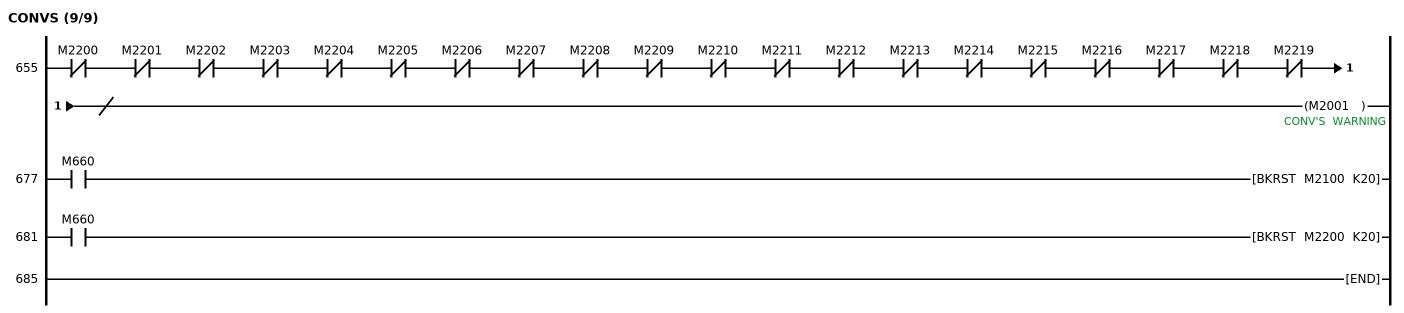
[picture p24: ladder of CONVS, rungs at steps 655 to 685]
655   LDI     M2200
      ANI     M2201
      ANI     M2202
      ANI     M2203
      ANI     M2204
      ANI     M2205
      ANI     M2206
      ANI     M2207
      ANI     M2208
      ANI     M2209
      ANI     M2210
      ANI     M2211
      ANI     M2212
      ANI     M2213
      ANI     M2214
      ANI     M2215
      ANI     M2216
      ANI     M2217
      ANI     M2218
      ANI     M2219
      INV
      OUT     M2001  ; CONV'S  WARNING
677   LD      M660
      BKRST   M2100 K20
681   LD      M660
      BKRST   M2200 K20
685   END
END_PROGRAM

PROGRAM CONV1
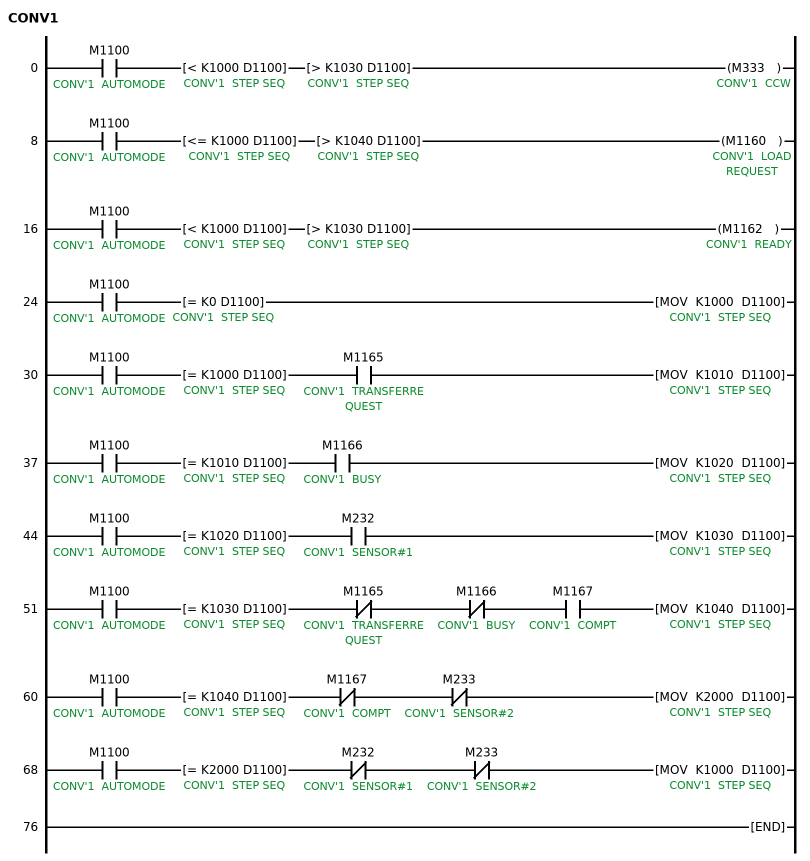
0     LD      M1100  ; CONV'1  AUTOMODE
      AND<    K1000 D1100  ; CONV'1  STEP SEQ
      AND>    K1030 D1100  ; CONV'1  STEP SEQ
      OUT     M333  ; CONV'1  CCW
8     LD      M1100  ; CONV'1  AUTOMODE
      AND<=   K1000 D1100  ; CONV'1  STEP SEQ
      AND>    K1040 D1100  ; CONV'1  STEP SEQ
      OUT     M1160  ; CONV'1  LOAD    REQUEST
16    LD      M1100  ; CONV'1  AUTOMODE
      AND<    K1000 D1100  ; CONV'1  STEP SEQ
      AND>    K1030 D1100  ; CONV'1  STEP SEQ
      OUT     M1162  ; CONV'1  READY
24    LD      M1100  ; CONV'1  AUTOMODE
      AND=    K0 D1100  ; CONV'1  STEP SEQ
      MOV     K1000 D1100
30    LD      M1100  ; CONV'1  AUTOMODE
      AND=    K1000 D1100  ; CONV'1  STEP SEQ
      AND     M1165  ; CONV'1  TRANSFERREQUEST
      MOV     K1010 D1100
37    LD      M1100  ; CONV'1  AUTOMODE
      AND=    K1010 D1100  ; CONV'1  STEP SEQ
      AND     M1166  ; CONV'1  BUSY
      MOV     K1020 D1100
44    LD      M1100  ; CONV'1  AUTOMODE
      AND=    K1020 D1100  ; CONV'1  STEP SEQ
      AND     M232  ; CONV'1  SENSOR#1
      MOV     K1030 D1100
51    LD      M1100  ; CONV'1  AUTOMODE
      AND=    K1030 D1100  ; CONV'1  STEP SEQ
      ANI     M1165  ; CONV'1  TRANSFERREQUEST
      ANI     M1166  ; CONV'1  BUSY
      AND     M1167  ; CONV'1  COMPT
      MOV     K1040 D1100
60    LD      M1100  ; CONV'1  AUTOMODE
      AND=    K1040 D1100  ; CONV'1  STEP SEQ
      ANI     M1167  ; CONV'1  COMPT
      ANI     M233  ; CONV'1  SENSOR#2
      MOV     K2000 D1100
68    LD      M1100  ; CONV'1  AUTOMODE
      AND=    K2000 D1100  ; CONV'1  STEP SEQ
      ANI     M232  ; CONV'1  SENSOR#1
      ANI     M233  ; CONV'1  SENSOR#2
      MOV     K1000 D1100
76    END
END_PROGRAM

PROGRAM CONV2
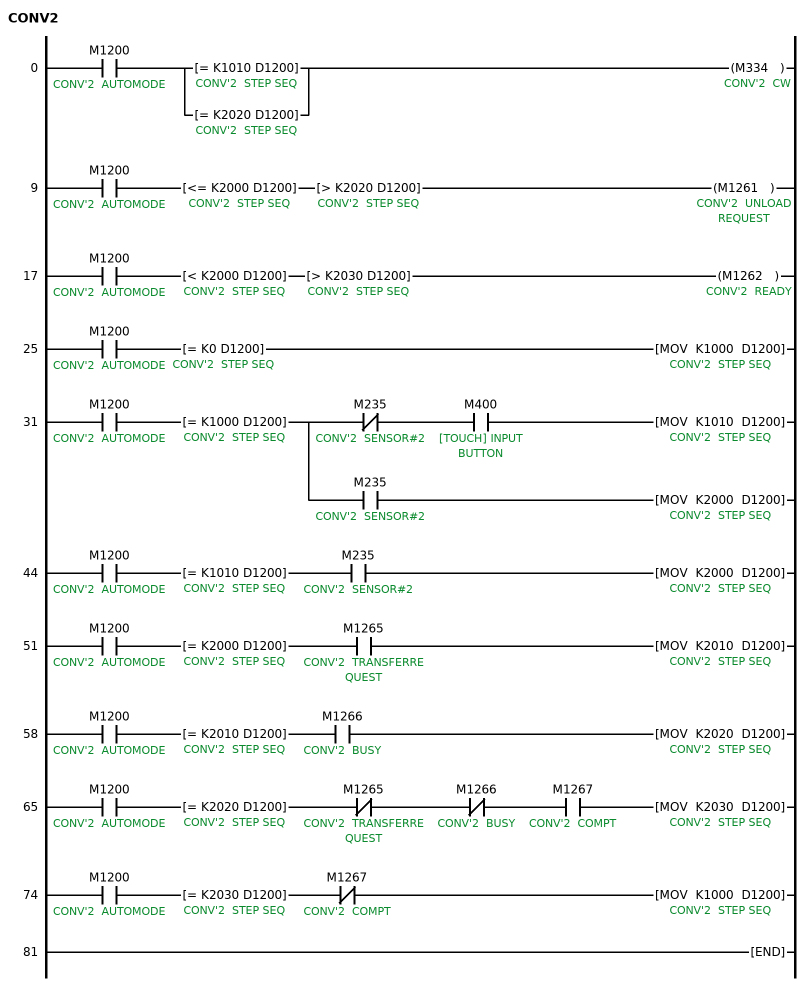
0     LD      M1200  ; CONV'2  AUTOMODE
      LD=     K1010 D1200  ; CONV'2  STEP SEQ
      OR=     K2020 D1200  ; CONV'2  STEP SEQ
      ANB
      OUT     M334  ; CONV'2  CW
9     LD      M1200  ; CONV'2  AUTOMODE
      AND<=   K2000 D1200  ; CONV'2  STEP SEQ
      AND>    K2020 D1200  ; CONV'2  STEP SEQ
      OUT     M1261  ; CONV'2  UNLOAD  REQUEST
17    LD      M1200  ; CONV'2  AUTOMODE
      AND<    K2000 D1200  ; CONV'2  STEP SEQ
      AND>    K2030 D1200  ; CONV'2  STEP SEQ
      OUT     M1262  ; CONV'2  READY
25    LD      M1200  ; CONV'2  AUTOMODE
      AND=    K0 D1200  ; CONV'2  STEP SEQ
      MOV     K1000 D1200
31    LD      M1200  ; CONV'2  AUTOMODE
      AND=    K1000 D1200  ; CONV'2  STEP SEQ
      MPS
      ANI     M235  ; CONV'2  SENSOR#2
      AND     M400  ; [TOUCH] INPUT   BUTTON
      MOV     K1010 D1200
      MPP
      AND     M235  ; CONV'2  SENSOR#2
      MOV     K2000 D1200
44    LD      M1200  ; CONV'2  AUTOMODE
      AND=    K1010 D1200  ; CONV'2  STEP SEQ
      AND     M235  ; CONV'2  SENSOR#2
      MOV     K2000 D1200
51    LD      M1200  ; CONV'2  AUTOMODE
      AND=    K2000 D1200  ; CONV'2  STEP SEQ
      AND     M1265  ; CONV'2  TRANSFERREQUEST
      MOV     K2010 D1200
58    LD      M1200  ; CONV'2  AUTOMODE
      AND=    K2010 D1200  ; CONV'2  STEP SEQ
      AND     M1266  ; CONV'2  BUSY
      MOV     K2020 D1200
65    LD      M1200  ; CONV'2  AUTOMODE
      AND=    K2020 D1200  ; CONV'2  STEP SEQ
      ANI     M1265  ; CONV'2  TRANSFERREQUEST
      ANI     M1266  ; CONV'2  BUSY
      AND     M1267  ; CONV'2  COMPT
      MOV     K2030 D1200
74    LD      M1200  ; CONV'2  AUTOMODE
      AND=    K2030 D1200  ; CONV'2  STEP SEQ
      ANI     M1267  ; CONV'2  COMPT
      MOV     K1000 D1200
81    END
END_PROGRAM

PROGRAM CONV3
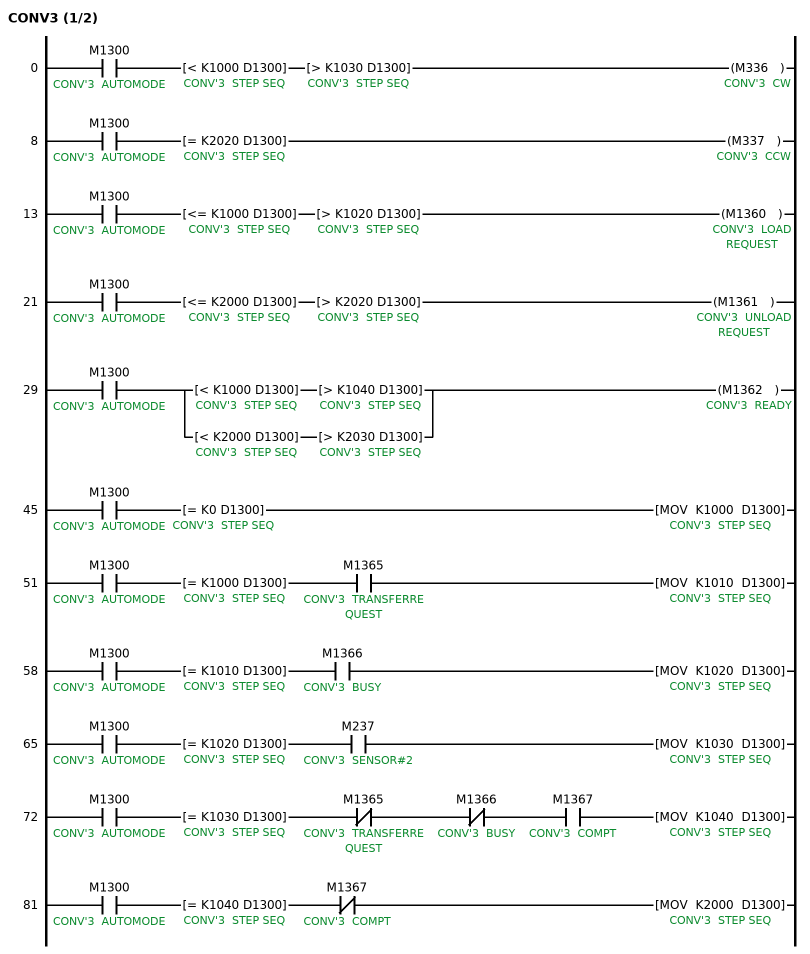
0     LD      M1300  ; CONV'3  AUTOMODE
      AND<    K1000 D1300  ; CONV'3  STEP SEQ
      AND>    K1030 D1300  ; CONV'3  STEP SEQ
      OUT     M336  ; CONV'3  CW
8     LD      M1300  ; CONV'3  AUTOMODE
      AND=    K2020 D1300  ; CONV'3  STEP SEQ
      OUT     M337  ; CONV'3  CCW
13    LD      M1300  ; CONV'3  AUTOMODE
      AND<=   K1000 D1300  ; CONV'3  STEP SEQ
      AND>    K1020 D1300  ; CONV'3  STEP SEQ
      OUT     M1360  ; CONV'3  LOAD    REQUEST
21    LD      M1300  ; CONV'3  AUTOMODE
      AND<=   K2000 D1300  ; CONV'3  STEP SEQ
      AND>    K2020 D1300  ; CONV'3  STEP SEQ
      OUT     M1361  ; CONV'3  UNLOAD  REQUEST
29    LD      M1300  ; CONV'3  AUTOMODE
      LD<     K1000 D1300  ; CONV'3  STEP SEQ
      AND>    K1040 D1300  ; CONV'3  STEP SEQ
      LD<     K2000 D1300  ; CONV'3  STEP SEQ
      AND>    K2030 D1300  ; CONV'3  STEP SEQ
      ORB
      ANB
      OUT     M1362  ; CONV'3  READY
45    LD      M1300  ; CONV'3  AUTOMODE
      AND=    K0 D1300  ; CONV'3  STEP SEQ
      MOV     K1000 D1300
51    LD      M1300  ; CONV'3  AUTOMODE
      AND=    K1000 D1300  ; CONV'3  STEP SEQ
      AND     M1365  ; CONV'3  TRANSFERREQUEST
      MOV     K1010 D1300
58    LD      M1300  ; CONV'3  AUTOMODE
      AND=    K1010 D1300  ; CONV'3  STEP SEQ
      AND     M1366  ; CONV'3  BUSY
      MOV     K1020 D1300
65    LD      M1300  ; CONV'3  AUTOMODE
      AND=    K1020 D1300  ; CONV'3  STEP SEQ
      AND     M237  ; CONV'3  SENSOR#2
      MOV     K1030 D1300
72    LD      M1300  ; CONV'3  AUTOMODE
      AND=    K1030 D1300  ; CONV'3  STEP SEQ
      ANI     M1365  ; CONV'3  TRANSFERREQUEST
      ANI     M1366  ; CONV'3  BUSY
      AND     M1367  ; CONV'3  COMPT
      MOV     K1040 D1300
81    LD      M1300  ; CONV'3  AUTOMODE
      AND=    K1040 D1300  ; CONV'3  STEP SEQ
      ANI     M1367  ; CONV'3  COMPT
      MOV     K2000 D1300
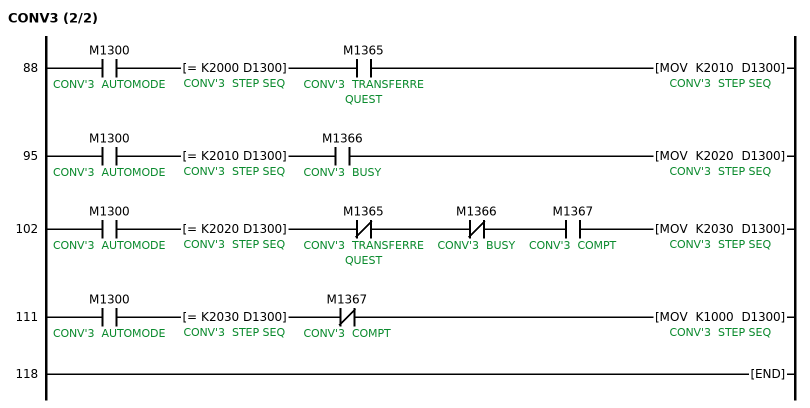
88    LD      M1300  ; CONV'3  AUTOMODE
      AND=    K2000 D1300  ; CONV'3  STEP SEQ
      AND     M1365  ; CONV'3  TRANSFERREQUEST
      MOV     K2010 D1300
95    LD      M1300  ; CONV'3  AUTOMODE
      AND=    K2010 D1300  ; CONV'3  STEP SEQ
      AND     M1366  ; CONV'3  BUSY
      MOV     K2020 D1300
102   LD      M1300  ; CONV'3  AUTOMODE
      AND=    K2020 D1300  ; CONV'3  STEP SEQ
      ANI     M1365  ; CONV'3  TRANSFERREQUEST
      ANI     M1366  ; CONV'3  BUSY
      AND     M1367  ; CONV'3  COMPT
      MOV     K2030 D1300
111   LD      M1300  ; CONV'3  AUTOMODE
      AND=    K2030 D1300  ; CONV'3  STEP SEQ
      ANI     M1367  ; CONV'3  COMPT
      MOV     K1000 D1300
118   END
END_PROGRAM

PROGRAM CONV4
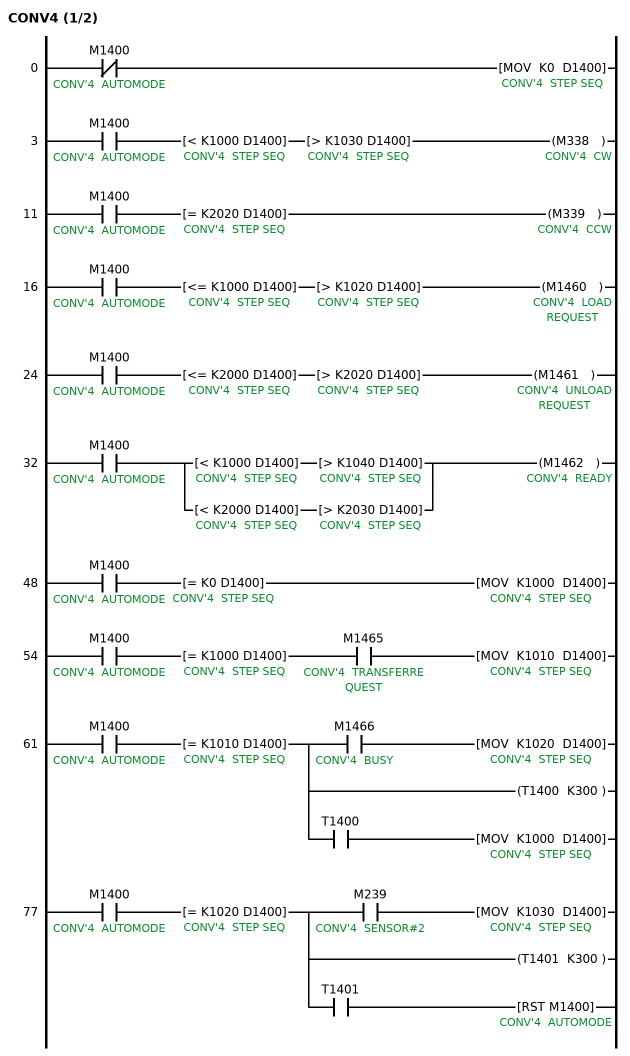
0     LDI     M1400  ; CONV'4  AUTOMODE
      MOV     K0 D1400  ; CONV'4  STEP SEQ
3     LD      M1400  ; CONV'4  AUTOMODE
      AND<    K1000 D1400  ; CONV'4  STEP SEQ
      AND>    K1030 D1400  ; CONV'4  STEP SEQ
      OUT     M338  ; CONV'4  CW
11    LD      M1400  ; CONV'4  AUTOMODE
      AND=    K2020 D1400  ; CONV'4  STEP SEQ
      OUT     M339  ; CONV'4  CCW
16    LD      M1400  ; CONV'4  AUTOMODE
      AND<=   K1000 D1400  ; CONV'4  STEP SEQ
      AND>    K1020 D1400  ; CONV'4  STEP SEQ
      OUT     M1460  ; CONV'4  LOAD    REQUEST
24    LD      M1400  ; CONV'4  AUTOMODE
      AND<=   K2000 D1400  ; CONV'4  STEP SEQ
      AND>    K2020 D1400  ; CONV'4  STEP SEQ
      OUT     M1461  ; CONV'4  UNLOAD  REQUEST
32    LD      M1400  ; CONV'4  AUTOMODE
      LD<     K1000 D1400  ; CONV'4  STEP SEQ
      AND>    K1040 D1400  ; CONV'4  STEP SEQ
      LD<     K2000 D1400  ; CONV'4  STEP SEQ
      AND>    K2030 D1400  ; CONV'4  STEP SEQ
      ORB
      ANB
      OUT     M1462  ; CONV'4  READY
48    LD      M1400  ; CONV'4  AUTOMODE
      AND=    K0 D1400  ; CONV'4  STEP SEQ
      MOV     K1000 D1400
54    LD      M1400  ; CONV'4  AUTOMODE
      AND=    K1000 D1400  ; CONV'4  STEP SEQ
      AND     M1465  ; CONV'4  TRANSFERREQUEST
      MOV     K1010 D1400
61    LD      M1400  ; CONV'4  AUTOMODE
      AND=    K1010 D1400  ; CONV'4  STEP SEQ
      MPS
      AND     M1466  ; CONV'4  BUSY
      MOV     K1020 D1400
      MPP
      OUT     T1400 K300
      AND     T1400
      MOV     K1000 D1400
77    LD      M1400  ; CONV'4  AUTOMODE
      AND=    K1020 D1400  ; CONV'4  STEP SEQ
      MPS
      AND     M239  ; CONV'4  SENSOR#2
      MOV     K1030 D1400
      MPP
      OUT     T1401 K300
      AND     T1401
      RST     M1400  ; CONV'4  AUTOMODE
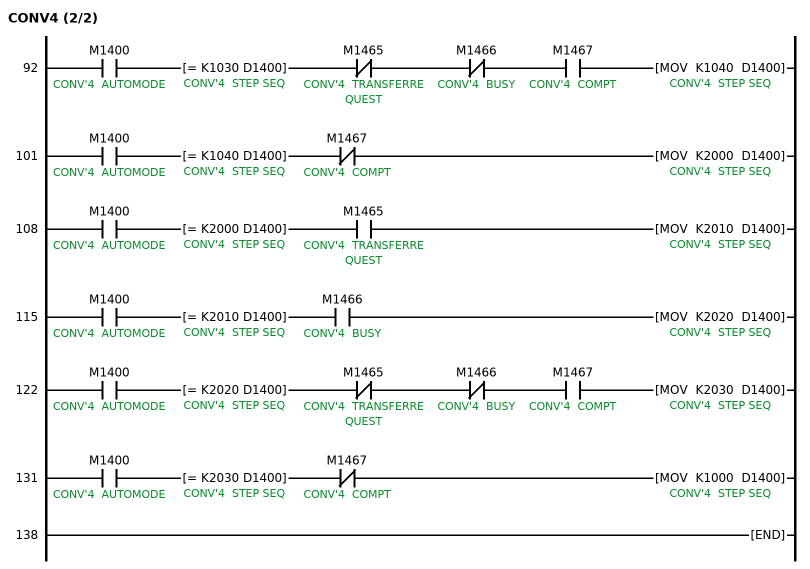
92    LD      M1400  ; CONV'4  AUTOMODE
      AND=    K1030 D1400  ; CONV'4  STEP SEQ
      ANI     M1465  ; CONV'4  TRANSFERREQUEST
      ANI     M1466  ; CONV'4  BUSY
      AND     M1467  ; CONV'4  COMPT
      MOV     K1040 D1400
101   LD      M1400  ; CONV'4  AUTOMODE
      AND=    K1040 D1400  ; CONV'4  STEP SEQ
      ANI     M1467  ; CONV'4  COMPT
      MOV     K2000 D1400
108   LD      M1400  ; CONV'4  AUTOMODE
      AND=    K2000 D1400  ; CONV'4  STEP SEQ
      AND     M1465  ; CONV'4  TRANSFERREQUEST
      MOV     K2010 D1400
115   LD      M1400  ; CONV'4  AUTOMODE
      AND=    K2010 D1400  ; CONV'4  STEP SEQ
      AND     M1466  ; CONV'4  BUSY
      MOV     K2020 D1400
122   LD      M1400  ; CONV'4  AUTOMODE
      AND=    K2020 D1400  ; CONV'4  STEP SEQ
      ANI     M1465  ; CONV'4  TRANSFERREQUEST
      ANI     M1466  ; CONV'4  BUSY
      AND     M1467  ; CONV'4  COMPT
      MOV     K2030 D1400
131   LD      M1400  ; CONV'4  AUTOMODE
      AND=    K2030 D1400  ; CONV'4  STEP SEQ
      ANI     M1467  ; CONV'4  COMPT
      MOV     K1000 D1400
138   END
END_PROGRAM

PROGRAM SERVO_ST
D1204 := 2 * 3 * 10; (*반지름 10을 사용하는 원 둘레를 구하는 공식*)
END_PROGRAM

FUNCTION_BLOCK SERVO_FB
VAR_INPUT
  SIMUL_MODE : BOOL;  (* SIMUL   MODE *)
  IN_SPEED : INT;  (* 1축G804 현재속도 *)
  IN_COMMAND : INT;  (* 1축G1500위치결정기동 *)
  IN_ERROR_RESET : INT;  (* 1축G1502에러레셋 *)
  IN_POSITION : INT;  (* 1축G1506현재변경값 *)
  IN_JOGSPEED : INT;  (* 1축G1518JOG속도 *)
END_VAR
VAR_OUTPUT
  OUT_POSITION : INT;  (* 1축G800 현재이송값 *)
  OUT_ERRORNUM : INT;  (* 1축G806 에러번호 *)
  OUT_SIGNAL : INT;  (* 1축G816 외부    입력신호 *)
  OUT_STATUS : INT;  (* 1축G817 현재상태 *)
END_VAR
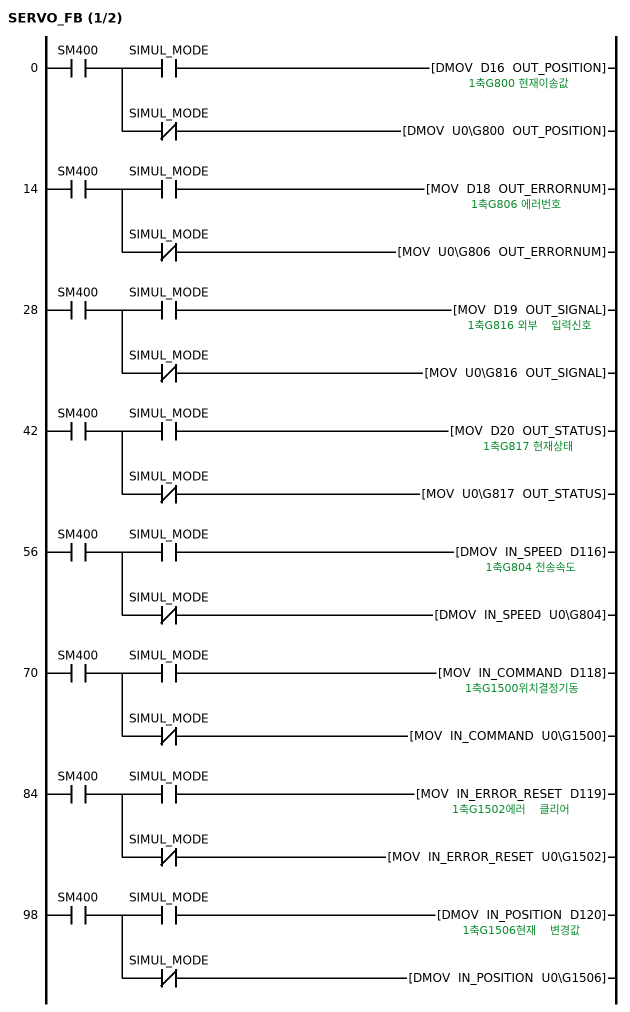
0     LD      SM400
      MPS
      AND     SIMUL_MODE
      DMOV    D16 OUT_POSITION  ; 1축G800 현재이송값
      MPP
      ANI     SIMUL_MODE
      DMOV    U0\G800 OUT_POSITION
14    LD      SM400
      MPS
      AND     SIMUL_MODE
      MOV     D18 OUT_ERRORNUM  ; 1축G806 에러번호
      MPP
      ANI     SIMUL_MODE
      MOV     U0\G806 OUT_ERRORNUM
28    LD      SM400
      MPS
      AND     SIMUL_MODE
      MOV     D19 OUT_SIGNAL  ; 1축G816 외부    입력신호
      MPP
      ANI     SIMUL_MODE
      MOV     U0\G816 OUT_SIGNAL
42    LD      SM400
      MPS
      AND     SIMUL_MODE
      MOV     D20 OUT_STATUS  ; 1축G817 현재상태
      MPP
      ANI     SIMUL_MODE
      MOV     U0\G817 OUT_STATUS
56    LD      SM400
      MPS
      AND     SIMUL_MODE
      DMOV    IN_SPEED D116  ; 1축G804 전송속도
      MPP
      ANI     SIMUL_MODE
      DMOV    IN_SPEED U0\G804
70    LD      SM400
      MPS
      AND     SIMUL_MODE
      MOV     IN_COMMAND D118  ; 1축G1500위치결정기동
      MPP
      ANI     SIMUL_MODE
      MOV     IN_COMMAND U0\G1500
84    LD      SM400
      MPS
      AND     SIMUL_MODE
      MOV     IN_ERROR_RESET D119  ; 1축G1502에러    클리어
      MPP
      ANI     SIMUL_MODE
      MOV     IN_ERROR_RESET U0\G1502
98    LD      SM400
      MPS
      AND     SIMUL_MODE
      DMOV    IN_POSITION D120  ; 1축G1506현재    변경값
      MPP
      ANI     SIMUL_MODE
      DMOV    IN_POSITION U0\G1506
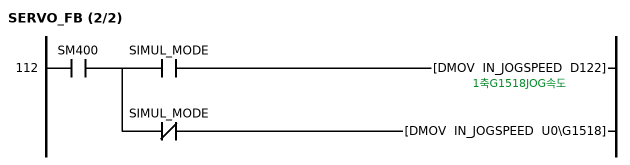
112   LD      SM400
      MPS
      AND     SIMUL_MODE
      DMOV    IN_JOGSPEED D122  ; 1축G1518JOG속도
      MPP
      ANI     SIMUL_MODE
      DMOV    IN_JOGSPEED U0\G1518
END_FUNCTION_BLOCK

FUNCTION_BLOCK MovePosition
VAR_INPUT
  SIMUL_MODE : BOOL;  (* SIMUL MODE *)
  IN_SPEED : INT;  (* 1축G804 현재속도 *)
  IN_COMMAND : INT;  (* [1축] 위치결정기동 *)
  IN_ERROR_RESET : INT;  (* [1축] 에러리셋 *)
  IN_POSITION : INT;  (* [1축] 현재변경값 *)
  IN_JOGSPEED : INT;  (* [1축] JOG속도 *)
END_VAR
VAR_OUTPUT
  OUT_POSITION : INT;  (* 1축G800 현재이송값 *)
  OUT_ERRORNUM : INT;  (* 1축G806 에러번호 *)
  OUT_SIGNAL : INT;  (* 1축G816 외부 입력신호 *)
  OUT-STATUS : INT;  (* 1축G817 현재상태 *)
END_VAR
END_FUNCTION_BLOCK

// device comments not shown above
M1070  ; CONV    S -> 1  READY
M1071  ; CONV    S -> 1  BUSY
M1110  ; CONV'1  CW
M1111  ; CONV'1  CW
M1115  ; CONV'1  CCW
M1116  ; CONV'1  CCW
M1210  ; CONV'2  CW
M1211  ; CONV'2  CW
